// SIMATIC S7-200 project (STEP 7-Micro/WIN), CPU 224 REL 02.01

ORGANIZATION_BLOCK MAIN:OB1
TITLE=程序是为汽车前照灯气密性测试设备设计的。包含手动和自动两种模式。系统应用于汽车制造或维修车间。
// 夹具装载前，夹具准备就绪传感器A 确认夹具位置正确，以确保装载顺利进行。夹具准备就绪传感器B 在夹具安装时提供额外的状态确认，以提高安全性。系统通过启动按钮启动自动测试流程，但前提是夹具完全就位传感器、夹具准备就绪传感器A 和夹具准备就绪传感器B 均确认夹具已正确放置，否则测试不会开始，以避免夹具未就位导致的测试失败或设备损坏。在自动模式下，夹具装载控制启动，由夹具装载定时器计时5个时间单位，确保夹具稳固安装。夹具装载完成后，测试压力控制阀打开，测试压力定时器计时5个时间单位以施加预设压力。压力达到后，压力传感器给出信号，泄漏检测控制启动，泄漏检测定时器计时15个时间单位，期间泄漏检测传感器监测是否有泄漏。若泄漏检测通过，测试合格指示灯点亮。测试结束后，夹具释放控制启动，夹具释放定时器计时15个时间单位，确保夹具安全卸载。操作员可通过停止按钮和紧急停止按钮控制流程停止。安全传感器检测到异常时，系统进入安全状态。系统支持手动模式和自动模式的切换，手动模式下可通过测试开始按钮和测试停止按钮控制测试。系统使用状态标志记录各阶段状态，确保流程可追溯。
// 控制系统设备包括气密试验机、夹具、气密性测试传感器、手动和自动模式开关、启动和停止按钮，可以说是较为复杂的程序了。
BEGIN
Network 1 // 网络标题
// 网络注释
LD     SM0.1
SLEN   " 06.12.1.4", VB0
?000
Network 2
LD     Q0.1
AN     I0.3
AN     I0.4
O      M0.0
A      I0.0
=      M0.0
Network 3
LDN    I0.1
A      I2.0
AN     M0.1
AN     M0.2
CALL   手动_2:SBR2
Network 4
LDN    I0.1
EU
AN     I1.0
A      I1.1
AN     I2.0
AN     M0.2
AN     M0.4
S      M0.1, 1
Network 5
LD     M0.1
AN     M0.2
AN     M0.4
AN     I2.0
CALL   夹具装载_0:SBR0
Network 6
LD     I0.1
EU
A      I1.0
AN     I1.1
AN     I2.0
AN     M0.1
AN     M0.4
S      M0.2, 1
Network 7
LD     M0.2
AN     M0.1
AN     M0.4
AN     I2.0
CALL   夹具释放_1:SBR1
Network 8
LD     I0.7
A      I1.0
AN     I1.1
AN     I2.0
AN     I0.1
AN     M0.1
AN     M0.2
CALL   自动_3:SBR3
Network 9
LD     M0.0
O      M0.3
O      M1.0
O      M1.1
A      SM0.5
=      Q0.0
END_ORGANIZATION_BLOCK

SUBROUTINE_BLOCK 夹具装载_0:SBR0
TITLE=子程序注释
BEGIN
Network 1 // 网络标题
// 网络注释
LD     M0.1
A      I1.1
A      I0.6
R      Q0.4, 1
Network 2
LD     M0.1
LD     I1.1
A      I0.7
O      I1.2
ALD
AN     M0.0
A      I0.0
AN     T103
R      Q0.2, 1
=      Q0.1
TON    T101, +5
Network 3
LD     I0.4
O      T101
A      M0.1
A      Q0.1
A      I1.1
A      I0.0
=      Q0.3
Network 4
LD     M0.1
A      I1.1
A      I1.2
TON    T102, +5
A      T102
R      Q0.6, 1
S      Q0.5, 1
Network 5
LD     M0.1
A      I1.0
LD     I1.2
O      Q0.2
ALD
ON     I0.0
LPS
TON    T103, +5
A      T103
AN     I0.5
S      Q0.2, 1
LPP
AN     Q0.0
AN     Q0.1
AN     I1.2
LD     Q0.2
O      I0.5
ALD
R      M0.1, 1
Network 6
LD     I0.7
A      I1.0
ON     I0.0
AN     Q0.0
AN     Q0.1
AN     Q0.2
R      M0.1, 1
END_SUBROUTINE_BLOCK

SUBROUTINE_BLOCK 夹具释放_1:SBR1
TITLE=
BEGIN
Network 1
LD     M0.2
AN     Q0.1
A      I1.0
A      I0.0
LPS
R      Q1.1, 1
TON    T103, +10
AN     Q0.1
=      Q1.0
=      Q2.3
LPP
LD     I1.3
O      Q0.7
ALD
AN     Q0.1
=      Q0.7
Network 2
LD     I0.0
A      T103
LPS
LD     Q0.7
A      I1.3
LDN    Q0.7
AN     I1.3
OLD
ALD
A      I1.4
AN     I3.2
=      L0.0
LPP
LD     Q0.7
AN     I1.3
ON     I1.4
O      I3.2
ALD
=      M0.3
Network 3
LD     M0.2
LD     L0.0
O      Q0.1
ALD
LDN    I1.1
ON     I0.6
ALD
AN     T104
A      I0.0
AN     M0.0
R      Q0.2, 1
=      Q0.1
TON    T101, +5
Network 4
LDN    I1.1
ON     I0.6
LD     T101
O      I0.4
ALD
A      M0.2
AN     M0.0
A      I0.0
=      Q0.3
Network 5
LD     M0.2
LDN    I1.1
ON     I0.6
ALD
A      I1.2
TON    T102, +5
A      T102
R      Q0.5, 1
S      Q0.6, 1
S      Q0.4, 1
Network 6
LD     M0.2
LD     I1.1
A      I0.6
O      M0.0
ALD
ON     I0.0
LPS
TON    T104, +5
A      T104
AN     I0.5
S      Q0.2, 1
LPP
AN     Q0.0
AN     Q0.1
LD     Q0.2
O      I0.5
ALD
R      M0.3, 1
R      M0.2, 1
END_SUBROUTINE_BLOCK

SUBROUTINE_BLOCK 手动_2:SBR2
TITLE=
BEGIN
Network 1
LD     I2.0
A      I2.1
A      I0.0
AN     M0.0
=      Q0.1
Network 2
LD     I2.0
A      I2.2
A      I0.0
=      Q0.2
Network 3
LD     I2.0
A      I2.3
A      I0.0
=      Q0.3
Network 4
LD     I2.0
A      I2.4
A      I0.0
=      Q0.4
Network 5
LD     I2.0
A      I2.5
A      I0.7
A      I1.2
A      I0.0
=      Q0.5
Network 6
LD     I2.0
A      I2.6
A      I0.7
A      I1.2
A      I0.0
=      Q0.6
Network 7
LD     I1.3
O      Q0.7
A      I2.0
A      I2.7
A      I1.2
A      I0.0
=      Q0.7
Network 8
LD     I2.0
A      I3.0
A      I1.2
A      I0.0
=      Q1.0
END_SUBROUTINE_BLOCK

SUBROUTINE_BLOCK 自动_3:SBR3
TITLE=
BEGIN
Network 1
LD     I0.2
EU
AN     I2.0
AN     I0.1
AN     M0.1
AN     M0.2
S      M0.4, 1
Network 2
LD     M0.4
EU
R      Q1.1, 1
Network 3
LD     I0.5
A      I0.2
O      Q0.1
AN     I2.0
A      M0.4
AN     M0.0
AN     T106
A      I0.0
LPS
R      Q0.2, 1
=      Q0.1
TON    T101, +5
A      I3.2
AN     T101
S      Q2.2, 1
LPP
A      T101
R      Q2.2, 1
Network 4
LD     M0.4
AN     M0.0
A      I0.0
LD     I0.4
O      T101
ALD
LPS
AN     M0.7
=      Q0.3
LPP
A      I1.2
TON    T102, +5
Network 5
LD     I1.3
O      Q0.7
A      M0.4
A      I1.2
A      T102
AN     M0.7
=      Q0.7
Network 6
LD     Q0.7
ON     I1.3
A      T102
A      I0.0
TON    T103, +15
Network 7
LD     M0.4
A      T102
LD     T103
ON     I1.3
O      T102
ALD
=      Q2.0
AN     I3.3
=      Q1.0
Network 8
LD     M0.4
A      Q2.0
A      I3.3
LPS
LD     I3.1
O      M0.6
ALD
LPS
S      M0.6, 1
TON    T104, +5
A      I3.1
AN     T104
S      Q2.2, 1
LPP
A      T104
R      Q2.2, 1
LPP
AN     I3.1
AN     M0.6
=      M1.0
Network 9
LD     M0.4
A      M0.6
A      T104
=      Q2.1
Network 10
LD     M0.4
A      Q2.1
LPS
A      I3.4
AN     I3.2
=      M0.7
LPP
AN     I3.4
A      I3.2
AN     Q1.1
=      M1.1
Network 11
LD     M0.4
A      M0.6
A      M0.7
LPS
TON    T105, +5
AN     T105
=      Q2.3
LPP
A      T105
S      M0.5, 1
S      Q1.1, 1
Network 12
LD     M0.4
LD     M0.5
O      M0.0
ALD
ON     I0.0
LPS
TON    T106, +5
A      T106
AN     I0.5
S      Q0.2, 1
LPP
AN     Q0.1
LD     Q0.2
O      I0.5
ALD
R      M0.5, 1
R      M0.6, 1
R      M0.7, 1
R      M0.4, 1
END_SUBROUTINE_BLOCK
